INTERFACE I_NodeAddedEvent EXTENDS I_Event

PROPERTY PUBLIC TargetNode : I_Node
GET
END_GET
END_PROPERTY

END_INTERFACE

(* stored: Version 1.1.0.1, ProductVersion 3.1.4024.12
   Itf I_NodeAddedEvent: Id {2b3e1ec7-33c7-4290-8fe4-794dd8aab3c5}
   Property TargetNode: Id {c912701a-dc7d-40a1-80a3-89f45cae7093}
   Get Get: Id {cd115d59-e4da-4411-80da-c75fa01bf282} *)
